Universal Robots PolyScope program: ayoo.urp

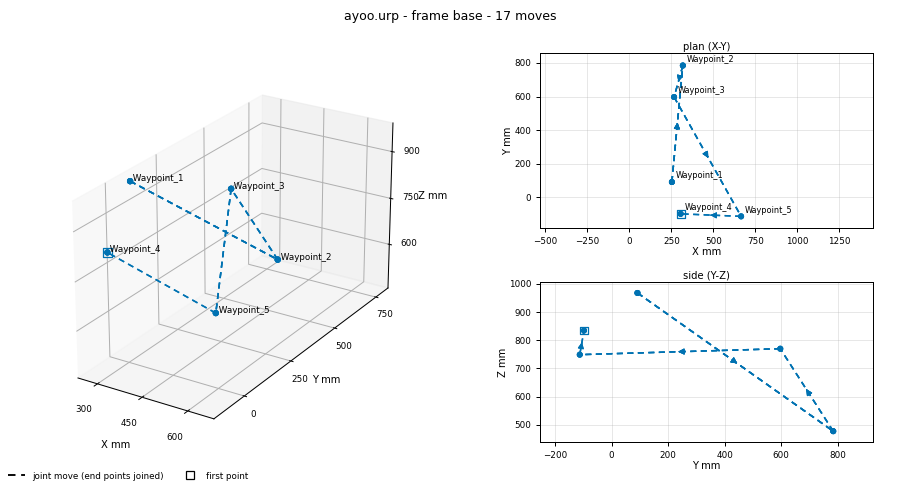
[picture p0: tool path of ayoo.urp in frame base, 17 of 26 moves have a stored position in this frame; points joined in program order, loops and branches not executed]
Program ayoo (createdIn=3.3.0.0 lastSavedIn=3.4.4.412 directory=/programs installation=default robotSerialNumber=2017356443)
Calibrated DH parameters: a=[0.000092, -0.116521, -0.182101, -0.000106, 0.000044, 0]; d=[0.089391, 255.189113, -82.629387, -172.449369, 0.094782, 0.082637]; alpha=[1.569598, 0.001603, 0.002015, 1.570234, -1.570307, 0]; deltaTheta=[-0.000017, 1.293309, -0.204843, -1.088417, 0.000036, -0.000078]
BeforeStart
  MoveJ speed 60 deg/s, acceleration 80 deg/s^2 (useActiveTCP=false)
    Waypoint Waypoint (Variable): variable(featureName=robopoint)
Robot Program (runOnlyOnce=false motionType=MoveJ speed=1.047198 acceleration=1.396263 useActiveTCP=false)
  Loop Counting (count=5) loopVariable(name=Loop_1)
    MoveJ speed 60 deg/s, acceleration 80 deg/s^2 (useActiveTCP=false)
      Waypoint Waypoint_4: TCP in base x=304.979 y=-97.943 z=834.545 mm, rx=-2.0857 ry=1.6975 rz=-0.5633 rad; joints [2.03, -87.238, -32.974, -117.268, 91.644, -9.379] deg
      Waypoint Waypoint (Variable): variable(featureName=robopoint)
